PROGRAM SetReset
VAR
	//reset dominant
	Set: BOOL;
	Reset: BOOL;
	Memory: BOOL;
	
	//set dominant
	
END_VAR

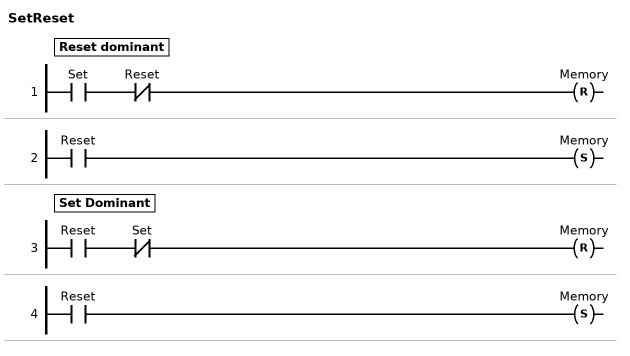
// NETWORK 1
// label: Reset dominant
Memory R= Set AND NOT Reset;

// NETWORK 2
Memory S= Reset;

// NETWORK 3
// label: Set Dominant
Memory R= Reset AND NOT Set;

// NETWORK 4
Memory S= Reset;

END_PROGRAM

(* stored: Version 1.1.0.1, ProductVersion 3.1.4024.10
   POU SetReset: Id {2e8131a0-91ab-440a-9946-2469cdbe8c3b}, SpecialFunc None *)
